{attribute 'qualified_only'}
VAR_GLOBAL
	// Communicatie tussen tasks
    coffeeReady : BOOL := FALSE;       // Wordt TRUE zodra koffie klaar is
    travelFinished : BOOL := FALSE;    // Wordt TRUE zodra je op school bent

    // Statussen
    travelState : INT := 0;            // Huidige stap in de reis
    coffeeState : INT := 0;            // Huidige stap in het koffietraject

    // Variabelen voor functie
    distanceToSchool : INT := 15;      // km
    avgSpeed : INT := 15;              // km/h
    travelTime : INT := 0;             // minuten, output van functie

END_VAR

(* stored: Version 1.1.0.1, ProductVersion 3.1.4024.15
   GVL GVL_Main: Id {6f43292f-8b76-43ac-a623-c9e4c390e1ad} *)
